(* Logix 5000 project; controller Generic 1768-L43 rev 15.6; software revision 15.01; part 6 of 10 *)
(* tags used below, declared in another part *)
   R04_OTE : DINT;
   AXIS_00 : AXIS_VIRTUAL;
   Axis_00_CMD : UDT_Axis_CMD;
   Axis_00_Data : UDT_Axis_Data;
   Axis_00_MI : UDT_Motion_Instructions;
   Axis_00_Status : UDT_Axis_Status;
   AXIS_01 : AXIS_SERVO_DRIVE;
   Axis_01_CMD : UDT_Axis_CMD;
   Axis_01_Data : UDT_Axis_Data;
   Axis_01_MI : UDT_Motion_Instructions;
   Axis_01_Status : UDT_Axis_Status;
   Axis_02_Status : UDT_Axis_Status;
   Axis_03_Status : UDT_Axis_Status;
   Axis_04_Status : UDT_Axis_Status;
   ClearFaultDelay : TIMER;
   GenericMachine_COND : UDT_Machine_COND;
   GUI_Axis_01_JogFwdREQ : BOOL;
   GUI_Axis_01_JogRevREQ : BOOL;
   GUI_Axis_01_ReferenceREQ : BOOL;
   GUI_Axis_02_JogFwdREQ : BOOL;
   GUI_Axis_02_JogRevREQ : BOOL;
   GUI_Axis_02_ReferenceREQ : BOOL;
   GUI_Axis_03_JogFwdREQ : BOOL;
   GUI_Axis_03_JogRevREQ : BOOL;
   GUI_Axis_03_ReferenceREQ : BOOL;
   GUI_Axis_04_JogFwdREQ : BOOL;
   GUI_Axis_04_JogRevREQ : BOOL;
   GUI_Axis_04_ReferenceREQ : BOOL;
   GUI_HoldRequest : BOOL;
   GUI_ManualControlRequest : BOOL;
   GUI_ReferenceREQ : BOOL;
   GUI_RunSPD_NI : DINT;
   GUI_StartRequest : BOOL;
   GUI_StopRequest : BOOL;
   ManualControl : BOOL;
   MotionGroup : MOTION_GROUP;
   PhaseTimout : UDT_PhaseTimeout;
   PowerUP_TMR : TIMER;
   PZ_GenericMachine_AUTO : PHASE;
   PZ_GenericMachine_MANUAL : PHASE;
(* P00_Control, continued *)

ROUTINE R03_PZ_Interface_AUTO   (* ladder *)
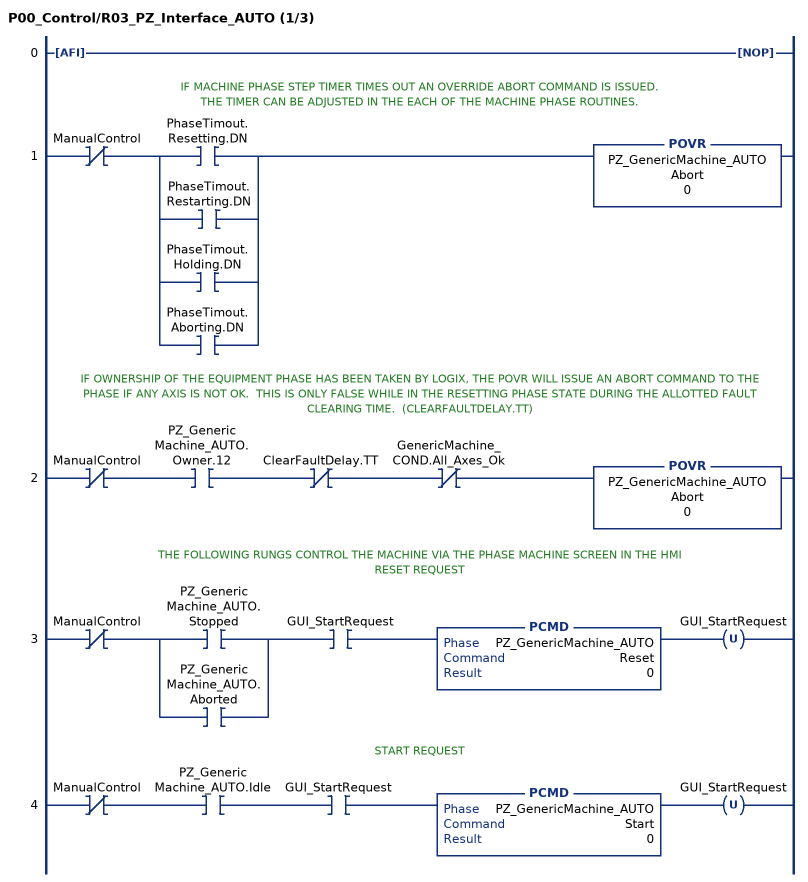
   0: AFI()NOP();
   // IF MACHINE PHASE STEP TIMER TIMES OUT AN OVERRIDE ABORT COMMAND IS ISSUED.
   // THE TIMER CAN BE ADJUSTED IN THE EACH OF THE MACHINE PHASE ROUTINES.
   1: XIO(ManualControl)[XIC(PhaseTimout.Resetting.DN) ,XIC(PhaseTimout.Restarting.DN) ,XIC(PhaseTimout.Holding.DN) ,XIC(PhaseTimout.Aborting.DN) ]POVR(PZ_GenericMachine_AUTO,Abort,0);
   // IF OWNERSHIP OF THE EQUIPMENT PHASE HAS BEEN TAKEN BY LOGIX, THE POVR WILL ISSUE AN ABORT COMMAND TO THE PHASE IF ANY AXIS IS NOT OK.  THIS IS ONLY FALSE WHILE IN THE RESETTING PHASE STATE DURING THE ALLOTTED FAULT CLEARING TIME.  (CLEARFAULTDELAY.TT)
   2: XIO(ManualControl)XIC(PZ_GenericMachine_AUTO.Owner.12)XIO(ClearFaultDelay.TT)XIO(GenericMachine_COND.All_Axes_Ok)POVR(PZ_GenericMachine_AUTO,Abort,0);
   // THE FOLLOWING RUNGS CONTROL THE MACHINE VIA THE PHASE MACHINE SCREEN IN THE HMI
   // RESET REQUEST
   3: XIO(ManualControl)[XIC(PZ_GenericMachine_AUTO.Stopped) ,XIC(PZ_GenericMachine_AUTO.Aborted) ]XIC(GUI_StartRequest)PCMD(PZ_GenericMachine_AUTO,Reset,0)OTU(GUI_StartRequest);
   // START REQUEST
   4: XIO(ManualControl)XIC(PZ_GenericMachine_AUTO.Idle)XIC(GUI_StartRequest)PCMD(PZ_GenericMachine_AUTO,Start,0)OTU(GUI_StartRequest);
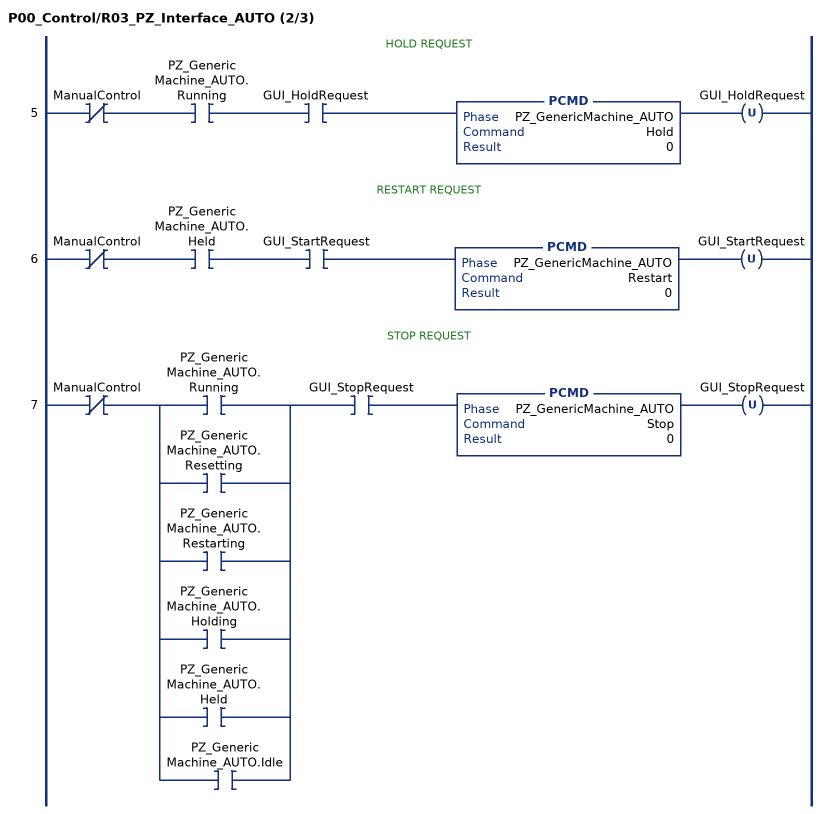
   // HOLD REQUEST
   5: XIO(ManualControl)XIC(PZ_GenericMachine_AUTO.Running)XIC(GUI_HoldRequest)PCMD(PZ_GenericMachine_AUTO,Hold,0)OTU(GUI_HoldRequest);
   // RESTART REQUEST
   6: XIO(ManualControl)XIC(PZ_GenericMachine_AUTO.Held)XIC(GUI_StartRequest)PCMD(PZ_GenericMachine_AUTO,Restart,0)OTU(GUI_StartRequest);
   // STOP REQUEST
   7: XIO(ManualControl)[XIC(PZ_GenericMachine_AUTO.Running) ,XIC(PZ_GenericMachine_AUTO.Resetting) ,XIC(PZ_GenericMachine_AUTO.Restarting) ,XIC(PZ_GenericMachine_AUTO.Holding) ,XIC(PZ_GenericMachine_AUTO.Held) ,XIC(PZ_GenericMachine_AUTO.Idle) ]XIC(GUI_StopRequest)PCMD(PZ_GenericMachine_AUTO,Stop,0)OTU(GUI_StopRequest);
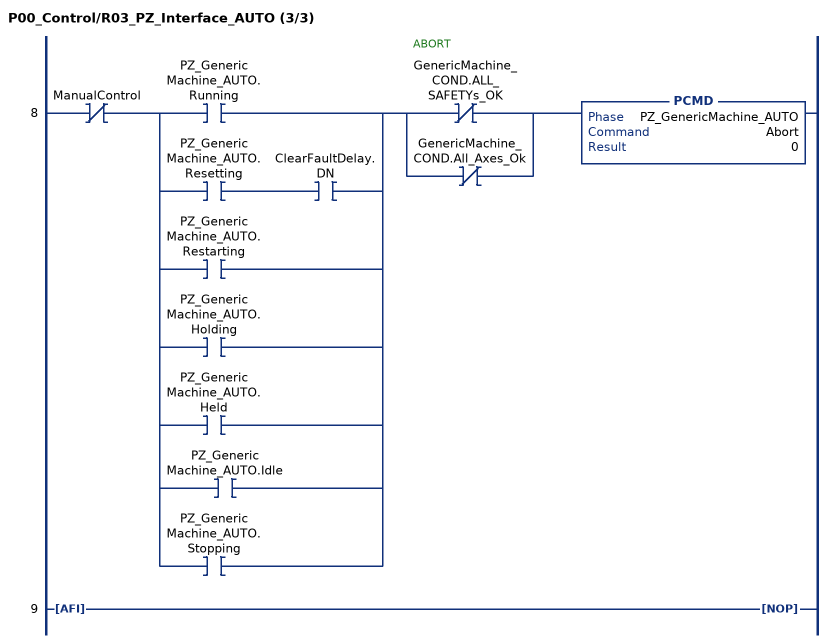
   // ABORT
   8: XIO(ManualControl)[XIC(PZ_GenericMachine_AUTO.Running) ,XIC(PZ_GenericMachine_AUTO.Resetting) XIC(ClearFaultDelay.DN) ,XIC(PZ_GenericMachine_AUTO.Restarting) ,XIC(PZ_GenericMachine_AUTO.Holding) ,XIC(PZ_GenericMachine_AUTO.Held) ,XIC(PZ_GenericMachine_AUTO.Idle) ,XIC(PZ_GenericMachine_AUTO.Stopping) ][XIO(GenericMachine_COND.ALL_SAFETYs_OK) ,XIO(GenericMachine_COND.All_Axes_Ok) ]PCMD(PZ_GenericMachine_AUTO,Abort,0);
   9: AFI()NOP();
END_ROUTINE

ROUTINE R04_PZ_Interface_MANUAL   (* ladder *)
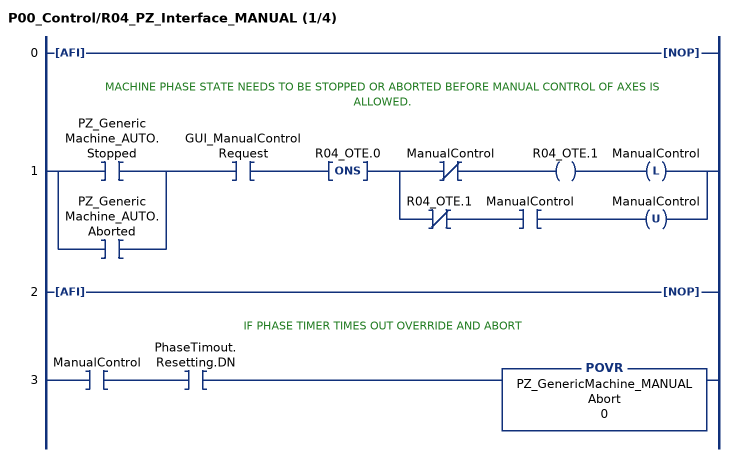
   0: AFI()NOP();
   // MACHINE PHASE STATE NEEDS TO BE STOPPED OR ABORTED BEFORE MANUAL CONTROL OF AXES IS ALLOWED.
   1: [XIC(PZ_GenericMachine_AUTO.Stopped) ,XIC(PZ_GenericMachine_AUTO.Aborted) ]XIC(GUI_ManualControlRequest)ONS(R04_OTE.0)[XIO(ManualControl) OTE(R04_OTE.1) OTL(ManualControl) ,XIO(R04_OTE.1) XIC(ManualControl) OTU(ManualControl) ];
   2: AFI()NOP();
   // IF PHASE TIMER TIMES OUT OVERRIDE AND ABORT
   3: XIC(ManualControl)XIC(PhaseTimout.Resetting.DN)POVR(PZ_GenericMachine_MANUAL,Abort,0);
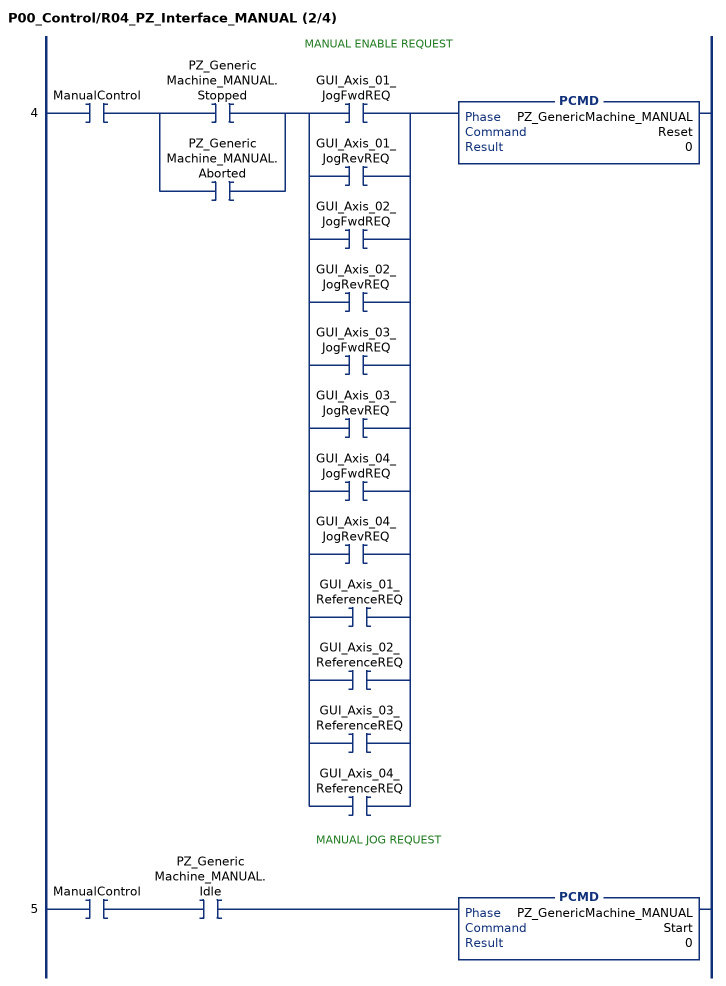
   // MANUAL ENABLE REQUEST
   4: XIC(ManualControl)[XIC(PZ_GenericMachine_MANUAL.Stopped) ,XIC(PZ_GenericMachine_MANUAL.Aborted) ][XIC(GUI_Axis_01_JogFwdREQ) ,XIC(GUI_Axis_01_JogRevREQ) ,XIC(GUI_Axis_02_JogFwdREQ) ,XIC(GUI_Axis_02_JogRevREQ) ,XIC(GUI_Axis_03_JogFwdREQ) ,XIC(GUI_Axis_03_JogRevREQ) ,XIC(GUI_Axis_04_JogFwdREQ) ,XIC(GUI_Axis_04_JogRevREQ) ,XIC(GUI_Axis_01_ReferenceREQ) ,XIC(GUI_Axis_02_ReferenceREQ) ,XIC(GUI_Axis_03_ReferenceREQ) ,XIC(GUI_Axis_04_ReferenceREQ) ]PCMD(PZ_GenericMachine_MANUAL,Reset,0);
   // MANUAL JOG REQUEST
   5: XIC(ManualControl)XIC(PZ_GenericMachine_MANUAL.Idle)PCMD(PZ_GenericMachine_MANUAL,Start,0);
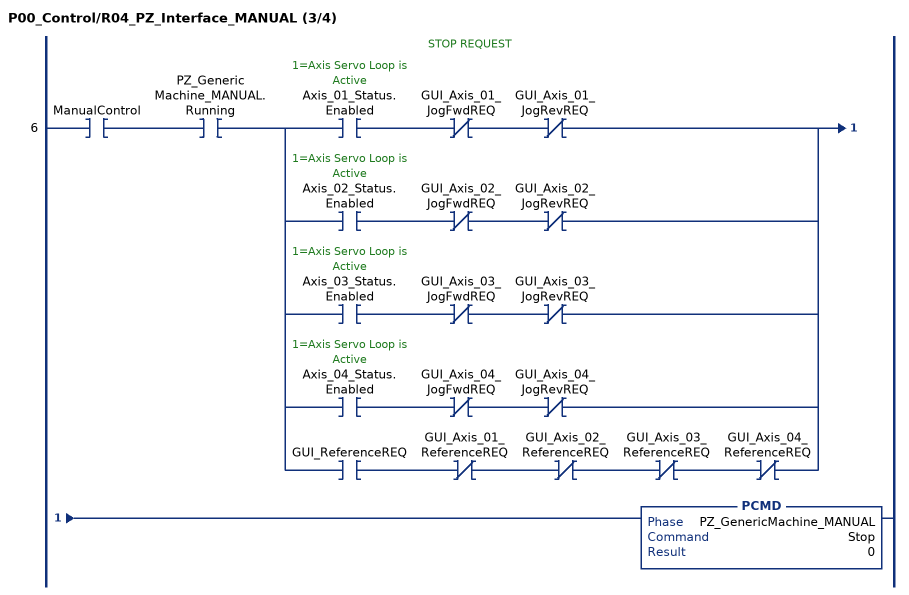
   // STOP REQUEST
   6: XIC(ManualControl)XIC(PZ_GenericMachine_MANUAL.Running)[XIC(Axis_01_Status.Enabled) XIO(GUI_Axis_01_JogFwdREQ) XIO(GUI_Axis_01_JogRevREQ) ,XIC(Axis_02_Status.Enabled) XIO(GUI_Axis_02_JogFwdREQ) XIO(GUI_Axis_02_JogRevREQ) ,XIC(Axis_03_Status.Enabled) XIO(GUI_Axis_03_JogFwdREQ) XIO(GUI_Axis_03_JogRevREQ) ,XIC(Axis_04_Status.Enabled) XIO(GUI_Axis_04_JogFwdREQ) XIO(GUI_Axis_04_JogRevREQ) ,XIC(GUI_ReferenceREQ) XIO(GUI_Axis_01_ReferenceREQ) XIO(GUI_Axis_02_ReferenceREQ) XIO(GUI_Axis_03_ReferenceREQ) XIO(GUI_Axis_04_ReferenceREQ) ]PCMD(PZ_GenericMachine_MANUAL,Stop,0);
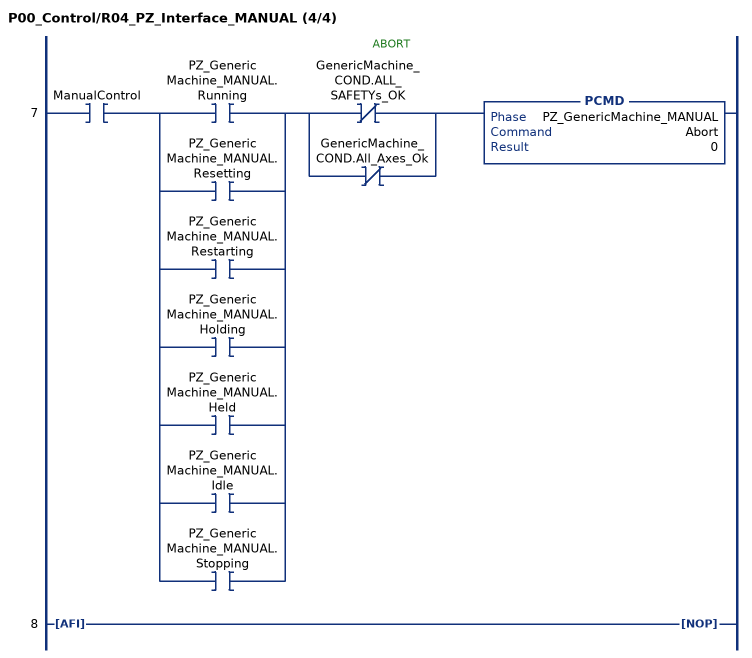
   // ABORT
   7: XIC(ManualControl)[XIC(PZ_GenericMachine_MANUAL.Running) ,XIC(PZ_GenericMachine_MANUAL.Resetting) ,XIC(PZ_GenericMachine_MANUAL.Restarting) ,XIC(PZ_GenericMachine_MANUAL.Holding) ,XIC(PZ_GenericMachine_MANUAL.Held) ,XIC(PZ_GenericMachine_MANUAL.Idle) ,XIC(PZ_GenericMachine_MANUAL.Stopping) ][XIO(GenericMachine_COND.ALL_SAFETYs_OK) ,XIO(GenericMachine_COND.All_Axes_Ok) ]PCMD(PZ_GenericMachine_MANUAL,Abort,0);
   8: AFI()NOP();
END_ROUTINE
END_PROGRAM

PROGRAM P01_AXIS_00   (* main routine R00_Dispatch *)
VAR
   Motion_Groups : ALIAS FOR MotionGroup;
   Servo_Axis : ALIAS FOR AXIS_00;
   Servo_CMD : ALIAS FOR Axis_00_CMD;
   Servo_DATA : ALIAS FOR Axis_00_Data;
   Servo_MI : ALIAS FOR Axis_00_MI;
   Servo_STATUS : ALIAS FOR Axis_00_Status;
END_VAR

ROUTINE R00_Dispatch   (* ladder *)
// THE DISPATCH ROUTINE CONTROLS EACH AXIS PROGRAM EXECUTION.
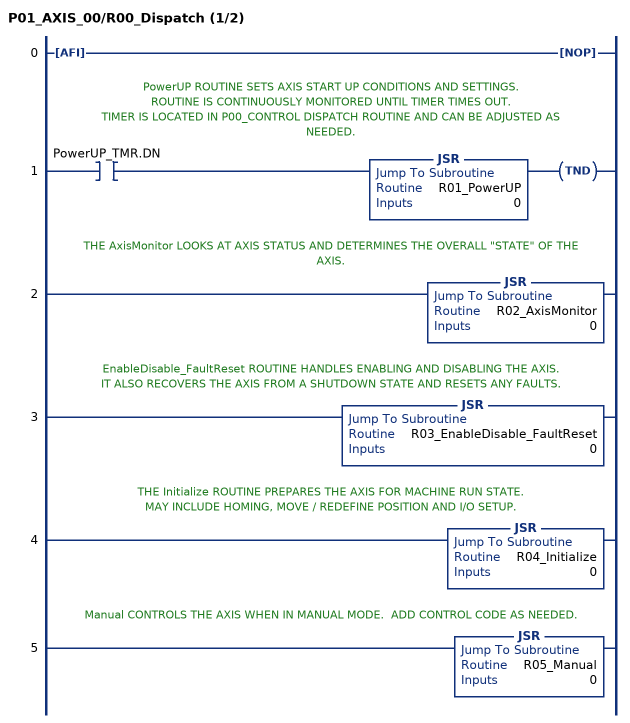
   0: AFI()NOP();
   // PowerUP ROUTINE SETS AXIS START UP CONDITIONS AND SETTINGS.
   // ROUTINE IS CONTINUOUSLY MONITORED UNTIL TIMER TIMES OUT.
   // TIMER IS LOCATED IN P00_CONTROL DISPATCH ROUTINE AND CAN BE ADJUSTED AS NEEDED.
   1: XIC(PowerUP_TMR.DN)JSR(R01_PowerUP,0)TND();
   // THE AxisMonitor LOOKS AT AXIS STATUS AND DETERMINES THE OVERALL "STATE" OF THE AXIS.
   2: JSR(R02_AxisMonitor,0);
   // EnableDisable_FaultReset ROUTINE HANDLES ENABLING AND DISABLING THE AXIS.
   // IT ALSO RECOVERS THE AXIS FROM A SHUTDOWN STATE AND RESETS ANY FAULTS.
   3: JSR(R03_EnableDisable_FaultReset,0);
   // THE Initialize ROUTINE PREPARES THE AXIS FOR MACHINE RUN STATE.
   // MAY INCLUDE HOMING, MOVE / REDEFINE POSITION AND I/O SETUP.
   4: JSR(R04_Initialize,0);
   // Manual CONTROLS THE AXIS WHEN IN MANUAL MODE.  ADD CONTROL CODE AS NEEDED.
   5: JSR(R05_Manual,0);
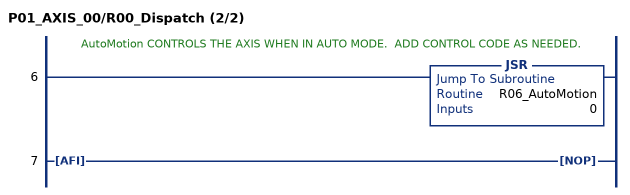
   // AutoMotion CONTROLS THE AXIS WHEN IN AUTO MODE.  ADD CONTROL CODE AS NEEDED.
   6: JSR(R06_AutoMotion,0);
   7: AFI()NOP();
END_ROUTINE

ROUTINE R01_PowerUP   (* ladder *)
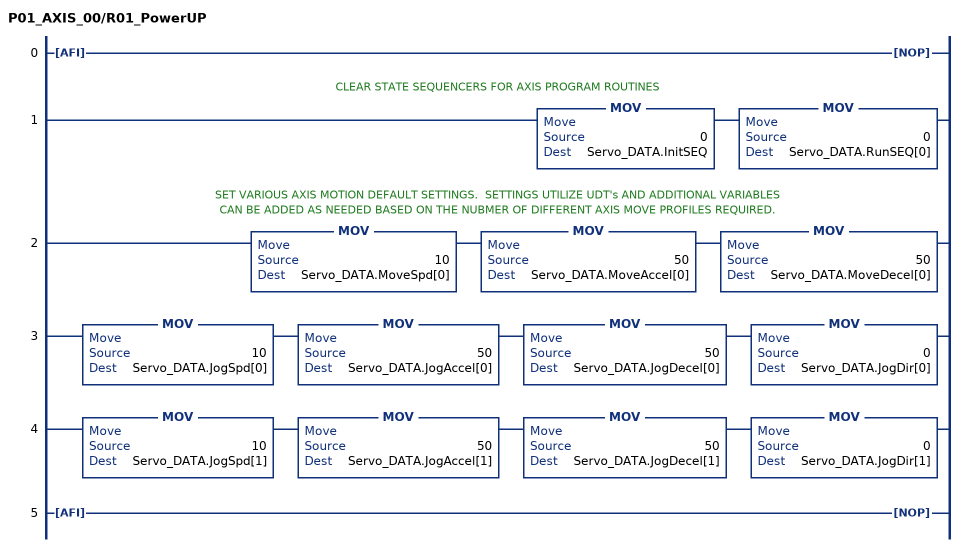
   0: AFI()NOP();
   // CLEAR STATE SEQUENCERS FOR AXIS PROGRAM ROUTINES
   1: MOV(0,Servo_DATA.InitSEQ)MOV(0,Servo_DATA.RunSEQ[0]);
   // SET VARIOUS AXIS MOTION DEFAULT SETTINGS.  SETTINGS UTILIZE UDT's AND ADDITIONAL VARIABLES
   // CAN BE ADDED AS NEEDED BASED ON THE NUBMER OF DIFFERENT AXIS MOVE PROFILES REQUIRED.
   2: MOV(10,Servo_DATA.MoveSpd[0])MOV(50,Servo_DATA.MoveAccel[0])MOV(50,Servo_DATA.MoveDecel[0]);
   3: MOV(10,Servo_DATA.JogSpd[0])MOV(50,Servo_DATA.JogAccel[0])MOV(50,Servo_DATA.JogDecel[0])MOV(0,Servo_DATA.JogDir[0]);
   4: MOV(10,Servo_DATA.JogSpd[1])MOV(50,Servo_DATA.JogAccel[1])MOV(50,Servo_DATA.JogDecel[1])MOV(0,Servo_DATA.JogDir[1]);
   5: AFI()NOP();
END_ROUTINE

ROUTINE R02_AxisMonitor   (* ladder *)
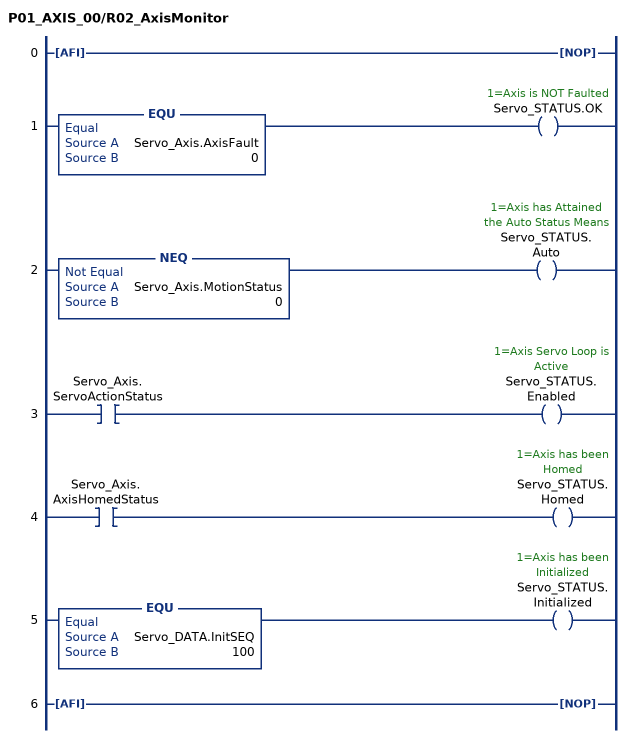
   0: AFI()NOP();
   1: EQU(Servo_Axis.AxisFault,0)OTE(Servo_STATUS.OK);
   2: NEQ(Servo_Axis.MotionStatus,0)OTE(Servo_STATUS.Auto);
   3: XIC(Servo_Axis.ServoActionStatus)OTE(Servo_STATUS.Enabled);
   4: XIC(Servo_Axis.AxisHomedStatus)OTE(Servo_STATUS.Homed);
   5: EQU(Servo_DATA.InitSEQ,100)OTE(Servo_STATUS.Initialized);
   6: AFI()NOP();
END_ROUTINE

ROUTINE R03_EnableDisable_FaultReset   (* ladder *)
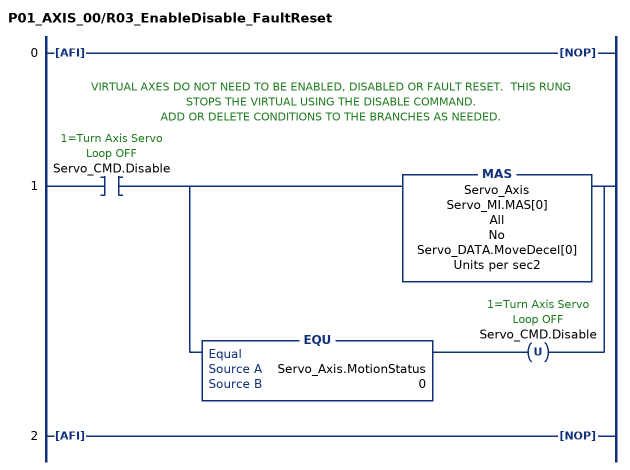
   0: AFI()NOP();
   // VIRTUAL AXES DO NOT NEED TO BE ENABLED, DISABLED OR FAULT RESET.  THIS RUNG STOPS THE VIRTUAL USING THE DISABLE COMMAND.
   // ADD OR DELETE CONDITIONS TO THE BRANCHES AS NEEDED.
   1: XIC(Servo_CMD.Disable)[MAS(Servo_Axis,Servo_MI.MAS[0],All,No,Servo_DATA.MoveDecel[0],Units per sec2) ,EQU(Servo_Axis.MotionStatus,0) OTU(Servo_CMD.Disable) ];
   2: AFI()NOP();
END_ROUTINE

ROUTINE R04_Initialize   (* ladder *)
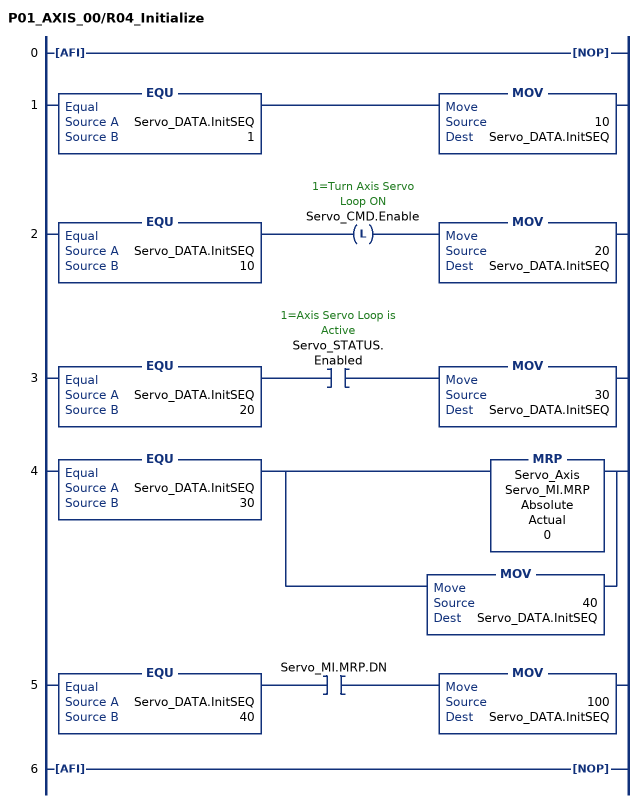
   0: AFI()NOP();
   1: EQU(Servo_DATA.InitSEQ,1)MOV(10,Servo_DATA.InitSEQ);
   2: EQU(Servo_DATA.InitSEQ,10)OTL(Servo_CMD.Enable)MOV(20,Servo_DATA.InitSEQ);
   3: EQU(Servo_DATA.InitSEQ,20)XIC(Servo_STATUS.Enabled)MOV(30,Servo_DATA.InitSEQ);
   4: EQU(Servo_DATA.InitSEQ,30)[MRP(Servo_Axis,Servo_MI.MRP,Absolute,Actual,0) ,MOV(40,Servo_DATA.InitSEQ) ];
   5: EQU(Servo_DATA.InitSEQ,40)XIC(Servo_MI.MRP.DN)MOV(100,Servo_DATA.InitSEQ);
   6: AFI()NOP();
END_ROUTINE

ROUTINE R05_Manual   (* ladder *)
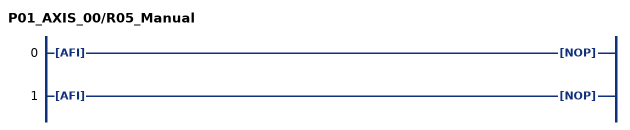
   0: AFI()NOP();
   1: AFI()NOP();
END_ROUTINE

ROUTINE R06_AutoMotion   (* ladder *)
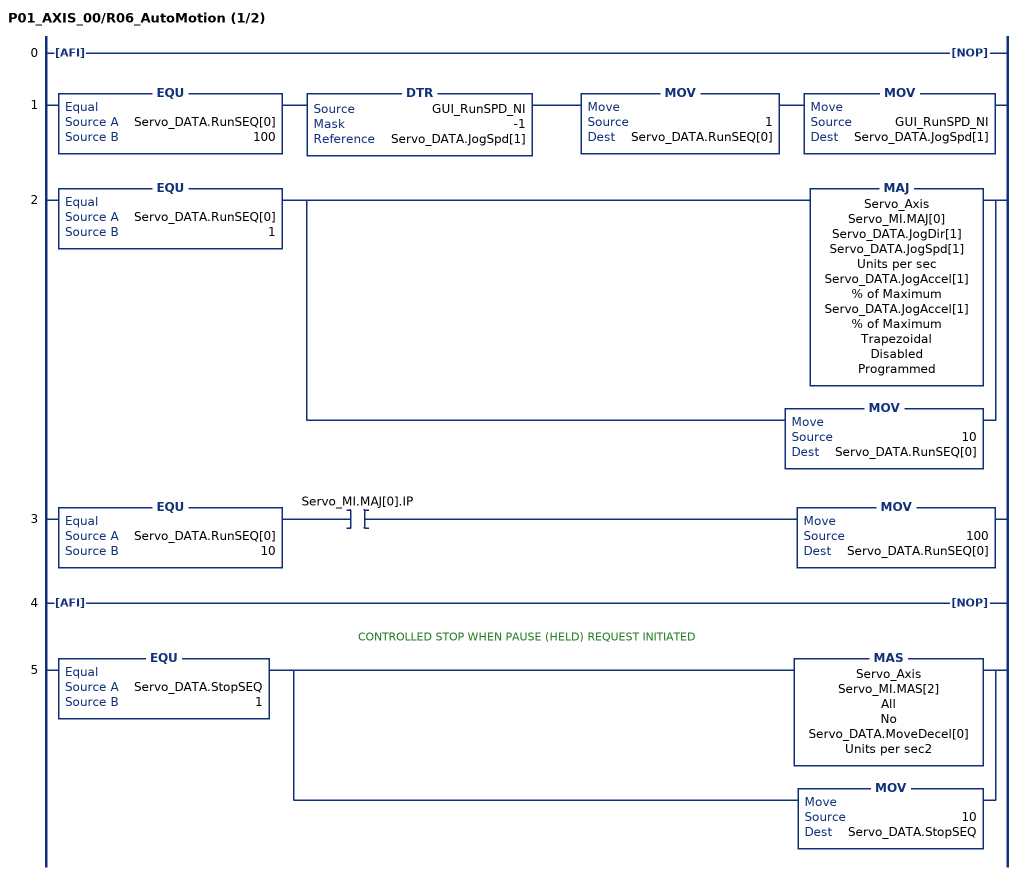
   0: AFI()NOP();
   1: EQU(Servo_DATA.RunSEQ[0],100)DTR(GUI_RunSPD_NI,-1,Servo_DATA.JogSpd[1])MOV(1,Servo_DATA.RunSEQ[0])MOV(GUI_RunSPD_NI,Servo_DATA.JogSpd[1]);
   2: EQU(Servo_DATA.RunSEQ[0],1)[MAJ(Servo_Axis,Servo_MI.MAJ[0],Servo_DATA.JogDir[1],Servo_DATA.JogSpd[1],Units per sec,Servo_DATA.JogAccel[1],% of Maximum,Servo_DATA.JogAccel[1],% of Maximum,Trapezoidal,Disabled,Programmed) ,MOV(10,Servo_DATA.RunSEQ[0]) ];
   3: EQU(Servo_DATA.RunSEQ[0],10)XIC(Servo_MI.MAJ[0].IP)MOV(100,Servo_DATA.RunSEQ[0]);
   4: AFI()NOP();
   // CONTROLLED STOP WHEN PAUSE (HELD) REQUEST INITIATED
   5: EQU(Servo_DATA.StopSEQ,1)[MAS(Servo_Axis,Servo_MI.MAS[2],All,No,Servo_DATA.MoveDecel[0],Units per sec2) ,MOV(10,Servo_DATA.StopSEQ) ];
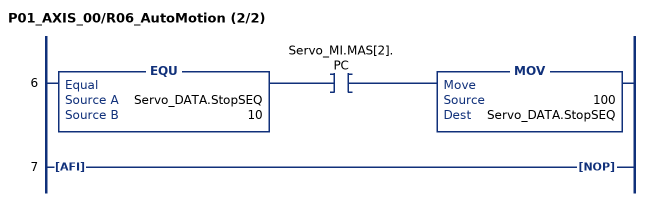
   6: EQU(Servo_DATA.StopSEQ,10)XIC(Servo_MI.MAS[2].PC)MOV(100,Servo_DATA.StopSEQ);
   7: AFI()NOP();
END_ROUTINE
END_PROGRAM

PROGRAM P02_AXIS_01   (* main routine R00_Dispatch *)
VAR
   Motion_Groups : ALIAS FOR MotionGroup;
   Servo_Axis : ALIAS FOR AXIS_01;
   Servo_CMD : ALIAS FOR Axis_01_CMD;
   Servo_DATA : ALIAS FOR Axis_01_Data;
   Servo_MI : ALIAS FOR Axis_01_MI;
   Servo_STATUS : ALIAS FOR Axis_01_Status;
END_VAR

ROUTINE R00_Dispatch   (* ladder *)
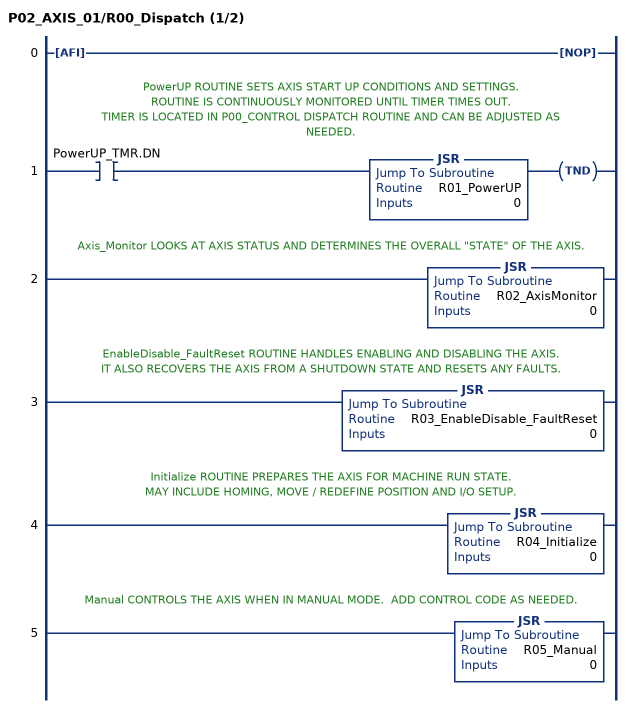
   0: AFI()NOP();
   // PowerUP ROUTINE SETS AXIS START UP CONDITIONS AND SETTINGS.
   // ROUTINE IS CONTINUOUSLY MONITORED UNTIL TIMER TIMES OUT.
   // TIMER IS LOCATED IN P00_CONTROL DISPATCH ROUTINE AND CAN BE ADJUSTED AS NEEDED.
   1: XIC(PowerUP_TMR.DN)JSR(R01_PowerUP,0)TND();
   // Axis_Monitor LOOKS AT AXIS STATUS AND DETERMINES THE OVERALL "STATE" OF THE AXIS.
   2: JSR(R02_AxisMonitor,0);
   // EnableDisable_FaultReset ROUTINE HANDLES ENABLING AND DISABLING THE AXIS.
   // IT ALSO RECOVERS THE AXIS FROM A SHUTDOWN STATE AND RESETS ANY FAULTS.
   3: JSR(R03_EnableDisable_FaultReset,0);
   // Initialize ROUTINE PREPARES THE AXIS FOR MACHINE RUN STATE.
   // MAY INCLUDE HOMING, MOVE / REDEFINE POSITION AND I/O SETUP.
   4: JSR(R04_Initialize,0);
   // Manual CONTROLS THE AXIS WHEN IN MANUAL MODE.  ADD CONTROL CODE AS NEEDED.
   5: JSR(R05_Manual,0);
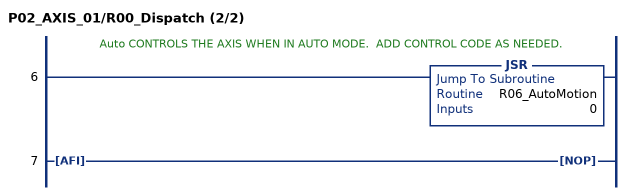
   // Auto CONTROLS THE AXIS WHEN IN AUTO MODE.  ADD CONTROL CODE AS NEEDED.
   6: JSR(R06_AutoMotion,0);
   7: AFI()NOP();
END_ROUTINE
